FUNCTION_BLOCK FB_Robot3R
VAR_INPUT
	Ts : LREAL := 0.01;
	bReset : BOOL;
	bEnableAll : BOOL;
	bEnableJoint : ARRAY [0..2] OF BOOL;
	eRobotModeCmd : E_RobotMode;
	fVelInput : ARRAY [0..2] OF LREAL;
	fPosInput : ARRAY [0..2] OF LREAL;
	fJointPositionOffset 	: ARRAY [0..2] OF LREAL;	
	fJointCalibrationOffset : ARRAY [0..2] OF LREAL;
END_VAR
VAR_OUTPUT
	eRobotMode : E_RobotMode;
	
	// Robot feedback
	q : ARRAY [0..2] OF LREAL;
	q_t : ARRAY [0..2] OF LREAL;
	tau : ARRAY [0..2] OF LREAL;
	
END_VAR
VAR
	bStop: BOOL;//Soft stop -> Ramp down first and then disables power
	bVelocityMode : BOOL;
	bPositionMode : BOOL;
	bPositionModeExecute : BOOL;

	// Setpoints
	qRef : ARRAY [0..2] OF LREAL;
	qRef_t : ARRAY [0..2] OF LREAL;
	qRef_tt : ARRAY [0..2] OF LREAL;	
	

	i : USINT;
	j : USINT;
	k : USINT;
	joints : ARRAY [0..2] OF FB_Joint;
	
	bAnyJointActive : BOOL;
	
	//Velcity of last timestamp
	fVelInputOld : ARRAY [0..2] OF LREAL;

END_VAR






IF eRobotModeCmd <> eRobotMode THEN
	CASE eRobotModeCmd OF
		 E_RobotMode.STOP:
		 
		 	bVelocityMode := FALSE;
			bPositionMode := FALSE;
			bPositionModeExecute := FALSE;
			
		 	eRobotMode := E_RobotMode.STOP;
			
		 E_RobotMode.ESTOP:
		 	

			bVelocityMode := FALSE;
			bPositionMode := FALSE;
			bPositionModeExecute := FALSE;
		 
		 	eRobotMode := E_RobotMode.ESTOP;
		 
		 E_RobotMode.POSITION:
		 	
			bVelocityMode := FALSE;
			bPositionMode := TRUE;
		 
		 	eRobotMode := E_RobotMode.POSITION;
		 
		 E_RobotMode.VELOCITY:
		 
			bVelocityMode := TRUE;
			bPositionMode := FALSE;
			bPositionModeExecute := FALSE;
		 	
		 	eRobotMode := E_RobotMode.VELOCITY;
	
	END_CASE	
END_IF


IF bReset THEN
	bEnableAll := FALSE;
END_IF

// E-stop mode
IF(eRobotMode = E_RobotMode.ESTOP OR NOT Safety.TS_I_Safety_EStopOK) THEN
	bEnableAll := FALSE;
	bReset := TRUE;	//to avoid error: the axis loss the enable signal while doing something
END_IF

// soft stop mode
IF(eRobotMode = E_RobotMode.STOP OR bStop) THEN
	bAnyJointActive := joints[0].bActive;
	FOR k:= 1 TO 2 DO
		bAnyJointActive := bAnyJointActive OR joints[k].bActive;	
	END_FOR
	
	IF NOT bAnyJointActive AND bStop THEN
		bEnableAll := FALSE;
	END_IF
END_IF

// position mode
IF(eRobotMode = E_RobotMode.POSITION) THEN
	positionMode();
// velocity mode
ELSIF(eRobotMode = E_RobotMode.VELOCITY) THEN
	velocityMode();
END_IF




// Execute joints
FOR j:= 0 TO 2 DO
	joints[j](
		bReset:=bReset,
		bEnable:=bEnableAll AND bEnableJoint[j],
		bStop:=bStop,
		bVelocityMode:=bVelocityMode,
		bPositionMode:=bPositionMode,
		bPositionModeExecute := bPositionModeExecute,
		qRef:=qRef[j],
		qRef_t := qRef_t[j],
		qRef_tt:=qRef_tt[j],
		fOffset := fJointPositionOffset[j] + fJointCalibrationOffset[j]
	);

	// Assign feedback data from joints
	q[j] := joints[j].q;
	q_t[j] := joints[j].q_t;
	tau[j] := joints[j].tau;
	
END_FOR

METHOD PRIVATE positionMode : BOOL
VAR_INPUT
	
END_VAR

FOR i:= 0 TO 2 DO
	IF joints[i].bActive THEN		
		// Set input based on velocity input u
		qRef[i] := fPosInput[i];
		qRef_t[i] := fVelInput[i];
		
	END_IF
	
END_FOR
END_METHOD

METHOD PRIVATE velocityMode : BOOL
VAR_INPUT
END_VAR
// Integrate position

FOR i:= 0 TO 2 DO
	qRef[i] := joints[i].q;
	IF joints[i].bActive THEN		
		// Set input based on velocity input u
		qRef[i] := qRef[i] + fVelInput[i]*Ts;
		qRef_t[i] := fVelInput[i];
		qRef_tt[i] := (fVelInput[i]-fVelInputOld[i])/(Ts);
		// Update old variable
		fVelInputOld[i] := fVelInput[i];
		
//	ELSE
//		qRef[i] := joints[i].q;
//		qRef_t[i] := 0;
//		qRef_tt[i] := 0;	
	END_IF
	
END_FOR
END_METHOD

END_FUNCTION_BLOCK

(* stored: Version 1.1.0.1, ProductVersion 3.1.4024.9
   POU FB_Robot3R: Id {ac314762-16df-47a2-b7b8-44cc8c775bfa}, SpecialFunc None
   Method positionMode: Id {f9d459a6-0feb-4986-b627-22787cb88f98}
   Method velocityMode: Id {125ad195-c68c-497a-bc79-95830c09961a} *)
